FUNCTION F_CheckAlarm
VAR_INPUT
	pTank : POINTER TO ST_Tank;
END_VAR
VAR
	fLevel : REAL := pTank^.fLevel;
	fTemperature : REAL := pTank^.fTemperature;
END_VAR


IF pTank <> 0 THEN
	IF fLevel > GVL.GC_MAX_LEVEL_PERCENT THEN
		pTank^.bLevelAlarm := TRUE;
	END_IF
	IF fTemperature > GVL.GC_MAX_TEMPERATURE THEN
		pTank^.bTemperatureAlarm := TRUE;
	END_IF
END_IF

END_FUNCTION

(* stored: Version 1.1.0.1, ProductVersion 3.1.4024.16
   POU F_CheckAlarm: Id {15ea5920-b8b7-4680-99e1-92531c40edad}, SpecialFunc None *)
